{attribute 'linkalways'}
{attribute 'hide_all_locals'}
FUNCTION_BLOCK ValueDt EXTENDS ValueDtRead IMPLEMENTS Value
VAR
END_VAR

METHOD SetFromType : BOOL
VAR_INPUT
	source : __SYSTEM.AnyType;
END_VAR
SetFromType := ConvertAnyType(source, thisAnyType);
END_METHOD

METHOD SetFromString : BOOL
VAR_INPUT
	value : T_MaxString;
END_VAR
thisValue := STRING_TO_DT(value);

SetFromString := TRUE;
END_METHOD

METHOD Set : BOOL
VAR_INPUT
	source : ANY;
END_VAR
Set := ConvertAnyType(source, thisAnyType);
END_METHOD

END_FUNCTION_BLOCK

(* stored: Version 1.1.0.1
   POU ValueDt: Id {3e038687-75e5-4204-a20d-291767981265}, SpecialFunc None
   Method SetFromType: Id {ae031a65-5fd9-4742-b9a1-44f3ddafdbcd}
   Method SetFromString: Id {cc78eb8f-94c8-4bc8-b823-7b9267d41580}
   Method Set: Id {1709bf2f-7212-4aeb-94f2-a2f5c5a75392} *)
